FUNCTION_BLOCK FB_AttenuatorSimulator
VAR_INPUT
	i_rRequestedAttenuation	:	REAL;
	i_stBPReadback	:	ST_BeamParams;
END_VAR
VAR_OUTPUT
	q_xFault	:	BOOL;
	q_rCurrentAttenuation	:	REAL;
END_VAR
VAR_IN_OUT
	Arbiter	:	FB_Arbiter; //Higher level arbiter from which upstream attenuation can be requested
END_VAR
VAR
	tonDelay	:	TON := (
		PT := T#3S
		);
END_VAR

// Really basic delay
tonDelay(IN := i_rRequestedAttenuation <> q_rCurrentAttenuation);

IF tonDelay.Q THEN
	q_rCurrentAttenuation := i_rRequestedAttenuation;
END_IF

END_FUNCTION_BLOCK

(* stored: Version 1.1.0.1, ProductVersion 3.1.4024.0
   POU FB_AttenuatorSimulator: Id {a3cc3cd5-f2d4-0113-3766-5daec5c567cb}, SpecialFunc None *)
